Omron Sysmac Studio project Duz_Zaman_Rolesi (Sysmac Studio 1.65.0.64007, StandardProject)

# Controller NX1P2: NX1P2-1040DT1 version 1.69
Task PrimaryTask (priority 4, period or condition 2000): Program0

VAR_GLOBAL
    BIO_Input_Bit_00 : BOOL;  (* at BuiltInIO://cpu/#0/Input_Bit_00 *)
    BIO_Input_Bit_01 : BOOL;  (* at BuiltInIO://cpu/#0/Input_Bit_01 *)
    BIO_Input_Bit_02 : BOOL;  (* at BuiltInIO://cpu/#0/Input_Bit_02 *)
    IN_Start_Button : BOOL;
    IN_Stop_Button : BOOL;
    IN_OptikSensor : BOOL;
    OUT_KonveyorMotor : BOOL;
    OUT_Motor1_Start : BOOL;
    OUT_Motor2_Start : BOOL;
    TON1_ET : TIME;
END_VAR

PROGRAM Program0
VAR
    Startt : BOOL;
    TON1 : TON;
    TON2 : TON;
    TON2_ET : TIME;
END_VAR
VAR_EXTERNAL
    BIO_Input_Bit_00 : BOOL;
    IN_Start_Button : BOOL;
    BIO_Input_Bit_01 : BOOL;
    IN_Stop_Button : BOOL;
    BIO_Input_Bit_02 : BOOL;
    IN_OptikSensor : BOOL;
    OUT_KonveyorMotor : BOOL;
    OUT_Motor1_Start : BOOL;
    OUT_Motor2_Start : BOOL;
    TON1_ET : TIME;
END_VAR

(* Section InOut: ladder, written here as Structured Text *)

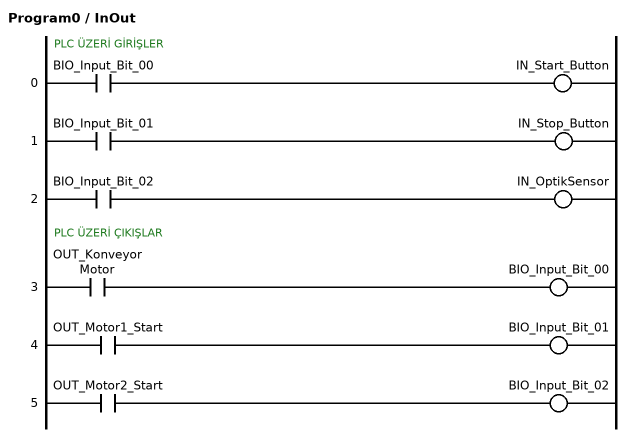
(* Rung 0: PLC ÜZERİ GİRİŞLER *)
IN_Start_Button := BIO_Input_Bit_00;
(* Rung 1 *)
IN_Stop_Button := BIO_Input_Bit_01;
(* Rung 2 *)
IN_OptikSensor := BIO_Input_Bit_02;
(* Rung 3: PLC ÜZERİ ÇIKIŞLAR *)
BIO_Input_Bit_00 := OUT_KonveyorMotor;
(* Rung 4 *)
BIO_Input_Bit_01 := OUT_Motor1_Start;
(* Rung 5 *)
BIO_Input_Bit_02 := OUT_Motor2_Start;

(* Section TON_Ornekleri: ladder, written here as Structured Text *)

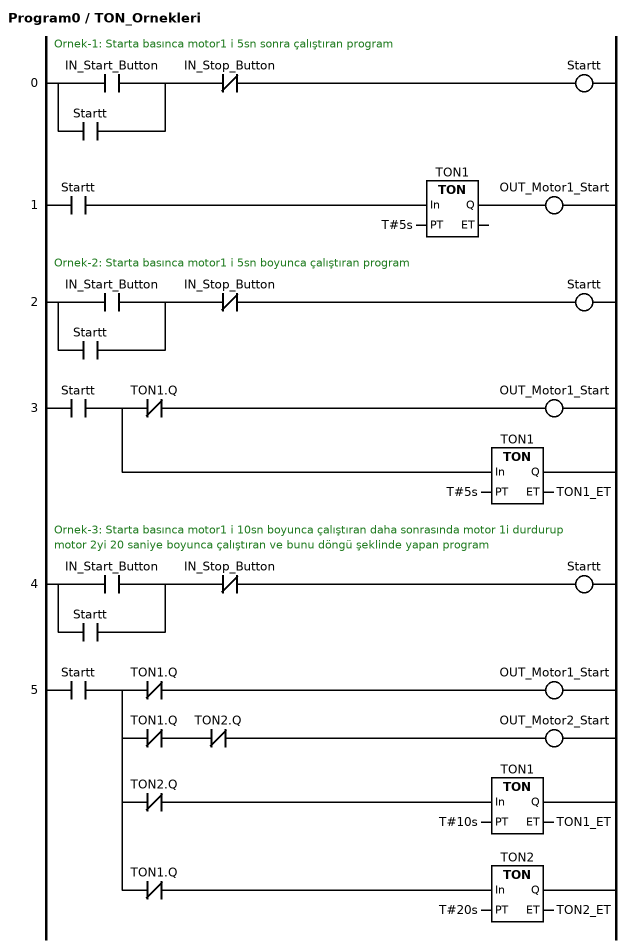
(* Rung 0: Ornek-1: Starta basınca motor1 i 5sn sonra çalıştıran program *)
Startt := (IN_Start_Button OR Startt) AND NOT IN_Stop_Button;
(* Rung 1 *)
TON1(In := Startt, PT := T#5s);
OUT_Motor1_Start := TON1.Q;
(* Rung 2: Ornek-2: Starta basınca motor1 i 5sn boyunca çalıştıran program *)
Startt := (IN_Start_Button OR Startt) AND NOT IN_Stop_Button;
(* Rung 3 *)
OUT_Motor1_Start := Startt AND NOT TON1.Q;
TON1(In := Startt, PT := T#5s, ET => TON1_ET);
(* Rung 4: Ornek-3: Starta basınca motor1 i 10sn boyunca çalıştıran daha sonrasında motor 1i durdurup motor 2yi 20 saniye boyunca çalıştıran ve bunu döngü şeklinde yapan program *)
Startt := (IN_Start_Button OR Startt) AND NOT IN_Stop_Button;
(* Rung 5 *)
OUT_Motor1_Start := Startt AND NOT TON1.Q;
OUT_Motor2_Start := Startt AND NOT TON1.Q AND NOT TON2.Q;
TON1(In := Startt AND NOT TON2.Q, PT := T#10s, ET => TON1_ET);
TON2(In := Startt AND NOT TON1.Q, PT := T#20s, ET => TON2_ET);
END_PROGRAM